(****************************************************************************************)
(*							Beckhoff Automation Poland									*)
(*								F_CLEAN_S2040	 v1.0									*)
(*									24.5.2011											*)
(*				Funkcja czyszcząca zawartość zmiennej typu ST_STRING_2040				*)
(*______________________________________________________________________________________*)
FUNCTION F_CLEAN_S2040 : ST_STRING_2040
VAR_INPUT
                VeryLongString: ST_STRING_2040;
END_VAR
VAR
                i: INT;                    (*iterator*)
END_VAR

FOR i := 1 TO 8 DO
                VeryLongString[i] := '$N';
END_FOR

END_FUNCTION

(* stored: Version 1.1.0.1, ProductVersion 3.1.4020.3
   POU F_CLEAN_S2040: Id {0029ef1c-7190-4cb8-9f78-ffa77f2b5c7b}, SpecialFunc None *)
